SYSTEM Skills
  (* Version 1.0, 2019-10-15, dorofeev *)
  APPLICATION SkillsApp
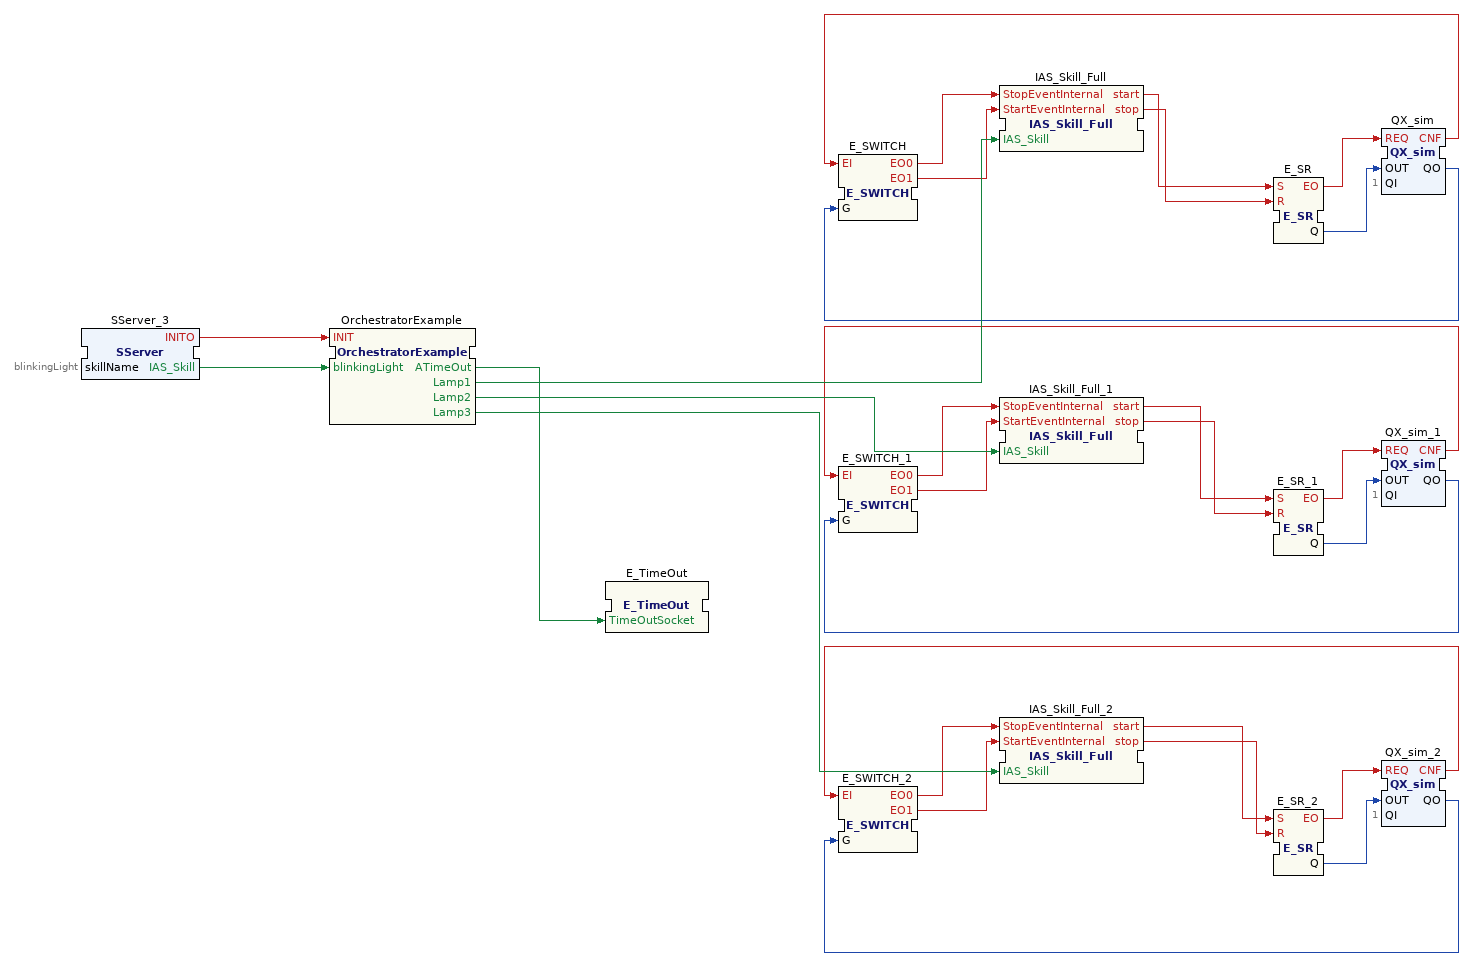
    FBS
      IAS_Skill_Full : IAS_Skill_Full;
      E_SR : E_SR;
      E_SWITCH : E_SWITCH;
      IAS_Skill_Full_1 : IAS_Skill_Full;
      E_SR_1 : E_SR;
      E_SWITCH_1 : E_SWITCH;
      IAS_Skill_Full_2 : IAS_Skill_Full;
      E_SR_2 : E_SR;
      E_SWITCH_2 : E_SWITCH;
      E_TimeOut : E_TimeOut;
      OrchestratorExample : OrchestratorExample;
    END_FBS
    SUBAPPS
      QX_sim : QX_sim(QI := 1);
      QX_sim_1 : QX_sim(QI := 1);
      QX_sim_2 : QX_sim(QI := 1);
      SServer_3 : SServer(skillName := blinkingLight);
    END_SUBAPPS
    EVENT_CONNECTIONS
      IAS_Skill_Full.start TO E_SR.S;
      IAS_Skill_Full.stop TO E_SR.R;
      E_SR.EO TO QX_sim.REQ;
      QX_sim.CNF TO E_SWITCH.EI;
      E_SWITCH.EO0 TO IAS_Skill_Full.StopEventInternal;
      E_SWITCH.EO1 TO IAS_Skill_Full.StartEventInternal;
      IAS_Skill_Full_1.start TO E_SR_1.S;
      E_SWITCH_1.EO0 TO IAS_Skill_Full_1.StopEventInternal;
      IAS_Skill_Full_1.stop TO E_SR_1.R;
      E_SWITCH_1.EO1 TO IAS_Skill_Full_1.StartEventInternal;
      QX_sim_1.CNF TO E_SWITCH_1.EI;
      E_SR_1.EO TO QX_sim_1.REQ;
      IAS_Skill_Full_2.start TO E_SR_2.S;
      E_SWITCH_2.EO0 TO IAS_Skill_Full_2.StopEventInternal;
      IAS_Skill_Full_2.stop TO E_SR_2.R;
      E_SWITCH_2.EO1 TO IAS_Skill_Full_2.StartEventInternal;
      QX_sim_2.CNF TO E_SWITCH_2.EI;
      E_SR_2.EO TO QX_sim_2.REQ;
      SServer_3.INITO TO OrchestratorExample.INIT;
    END_CONNECTIONS
    DATA_CONNECTIONS
      E_SR.Q TO QX_sim.OUT;
      QX_sim.QO TO E_SWITCH.G;
      E_SR_1.Q TO QX_sim_1.OUT;
      QX_sim_1.QO TO E_SWITCH_1.G;
      E_SR_2.Q TO QX_sim_2.OUT;
      QX_sim_2.QO TO E_SWITCH_2.G;
    END_CONNECTIONS
    ADAPTER_CONNECTIONS
      OrchestratorExample.ATimeOut TO E_TimeOut.TimeOutSocket;
      SServer_3.IAS_Skill TO OrchestratorExample.blinkingLight;
      OrchestratorExample.Lamp1 TO IAS_Skill_Full.IAS_Skill;
      OrchestratorExample.Lamp2 TO IAS_Skill_Full_1.IAS_Skill;
      OrchestratorExample.Lamp3 TO IAS_Skill_Full_2.IAS_Skill;
    END_CONNECTIONS
  END_APPLICATION
  APPLICATION test
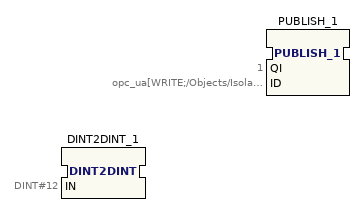
    FBS
      PUBLISH_1 : PUBLISH_1(QI := 1, ID := opc_ua[WRITE;/Objects/IsolatedTests/WRITEVariable]);
      DINT2DINT_1 : DINT2DINT(IN := DINT#12);
    END_FBS
  END_APPLICATION
  DEVICE skillConsumer : FORTE_PC(MGR_ID := "localhost:61499")
    {SET_ATTRIBUTE(Profile, HOLOBLOC)} (* device profile *)
    RESOURCE EMB_RES : EMB_RES
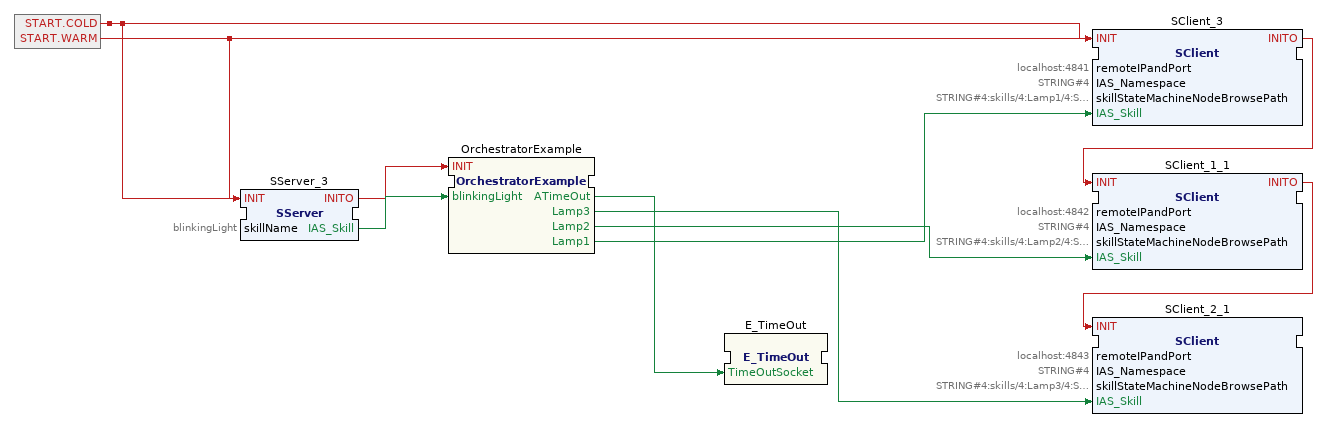
      FBS
        E_TimeOut : E_TimeOut;
        OrchestratorExample : OrchestratorExample;
      END_FBS
      SUBAPPS
        SServer_3 : SServer(skillName := blinkingLight);
        SClient_2_1 : SClient(remoteIPandPort := localhost:4843, IAS_Namespace := STRING#4, skillStateMachineNodeBrowsePath := STRING#4:skills/4:Lamp3/4:StateMachine/);
        SClient_3 : SClient(remoteIPandPort := localhost:4841, IAS_Namespace := STRING#4, skillStateMachineNodeBrowsePath := STRING#4:skills/4:Lamp1/4:StateMachine/);
        SClient_1_1 : SClient(remoteIPandPort := localhost:4842, IAS_Namespace := STRING#4, skillStateMachineNodeBrowsePath := STRING#4:skills/4:Lamp2/4:StateMachine/);
      END_SUBAPPS
      EVENT_CONNECTIONS
        SServer_3.INITO TO OrchestratorExample.INIT;
        START.COLD TO SServer_3.INIT;
        START.WARM TO SServer_3.INIT;
        SClient_1_1.INITO TO SClient_2_1.INIT;
        SClient_3.INITO TO SClient_1_1.INIT;
        START.COLD TO SClient_3.INIT;
        START.WARM TO SClient_3.INIT;
      END_CONNECTIONS
      ADAPTER_CONNECTIONS
        OrchestratorExample.ATimeOut TO E_TimeOut.TimeOutSocket;
        SServer_3.IAS_Skill TO OrchestratorExample.blinkingLight;
        OrchestratorExample.Lamp3 TO SClient_2_1.IAS_Skill;
        OrchestratorExample.Lamp2 TO SClient_1_1.IAS_Skill;
        OrchestratorExample.Lamp1 TO SClient_3.IAS_Skill;
      END_CONNECTIONS
    END_RESOURCE
  END_DEVICE
  DEVICE skillProvider1 : FORTE_PC(MGR_ID := "localhost:61500")
    {SET_ATTRIBUTE(Profile, HOLOBLOC)} (* device profile *)
    RESOURCE EMB_RES : EMB_RES
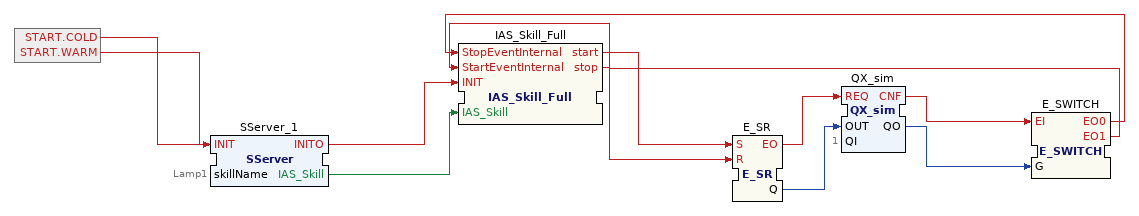
      FBS
        IAS_Skill_Full : IAS_Skill_Full;
        E_SWITCH : E_SWITCH;
        E_SR : E_SR;
      END_FBS
      SUBAPPS
        QX_sim : QX_sim(QI := 1);
        SServer_1 : SServer(skillName := Lamp1);
      END_SUBAPPS
      EVENT_CONNECTIONS
        QX_sim.CNF TO E_SWITCH.EI;
        E_SWITCH.EO0 TO IAS_Skill_Full.StopEventInternal;
        E_SWITCH.EO1 TO IAS_Skill_Full.StartEventInternal;
        IAS_Skill_Full.start TO E_SR.S;
        IAS_Skill_Full.stop TO E_SR.R;
        E_SR.EO TO QX_sim.REQ;
        START.COLD TO SServer_1.INIT;
        START.WARM TO SServer_1.INIT;
        SServer_1.INITO TO IAS_Skill_Full.INIT;
      END_CONNECTIONS
      DATA_CONNECTIONS
        QX_sim.QO TO E_SWITCH.G;
        E_SR.Q TO QX_sim.OUT;
      END_CONNECTIONS
      ADAPTER_CONNECTIONS
        SServer_1.IAS_Skill TO IAS_Skill_Full.IAS_Skill;
      END_CONNECTIONS
    END_RESOURCE
  END_DEVICE
  DEVICE skillProvider2 : FORTE_PC(MGR_ID := "localhost:61501")
    {SET_ATTRIBUTE(Profile, HOLOBLOC)} (* device profile *)
    RESOURCE EMB_RES : EMB_RES
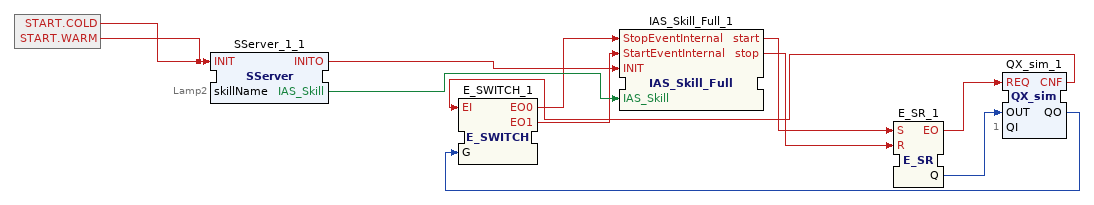
      FBS
        IAS_Skill_Full_1 : IAS_Skill_Full;
        E_SR_1 : E_SR;
        E_SWITCH_1 : E_SWITCH;
      END_FBS
      SUBAPPS
        QX_sim_1 : QX_sim(QI := 1);
        SServer_1_1 : SServer(skillName := Lamp2);
      END_SUBAPPS
      EVENT_CONNECTIONS
        IAS_Skill_Full_1.start TO E_SR_1.S;
        IAS_Skill_Full_1.stop TO E_SR_1.R;
        E_SR_1.EO TO QX_sim_1.REQ;
        QX_sim_1.CNF TO E_SWITCH_1.EI;
        E_SWITCH_1.EO0 TO IAS_Skill_Full_1.StopEventInternal;
        E_SWITCH_1.EO1 TO IAS_Skill_Full_1.StartEventInternal;
        START.COLD TO SServer_1_1.INIT;
        START.WARM TO SServer_1_1.INIT;
        SServer_1_1.INITO TO IAS_Skill_Full_1.INIT;
      END_CONNECTIONS
      DATA_CONNECTIONS
        E_SR_1.Q TO QX_sim_1.OUT;
        QX_sim_1.QO TO E_SWITCH_1.G;
      END_CONNECTIONS
      ADAPTER_CONNECTIONS
        SServer_1_1.IAS_Skill TO IAS_Skill_Full_1.IAS_Skill;
      END_CONNECTIONS
    END_RESOURCE
  END_DEVICE
  DEVICE skillProvider3 : FORTE_PC(MGR_ID := "localhost:61502")
    {SET_ATTRIBUTE(Profile, HOLOBLOC)} (* device profile *)
    RESOURCE EMB_RES : EMB_RES
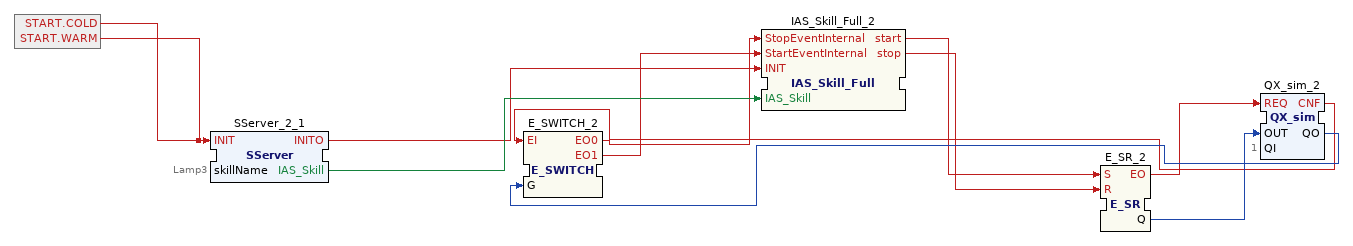
      FBS
        E_SWITCH_2 : E_SWITCH;
        E_SR_2 : E_SR;
        IAS_Skill_Full_2 : IAS_Skill_Full;
      END_FBS
      SUBAPPS
        QX_sim_2 : QX_sim(QI := 1);
        SServer_2_1 : SServer(skillName := Lamp3);
      END_SUBAPPS
      EVENT_CONNECTIONS
        E_SR_2.EO TO QX_sim_2.REQ;
        QX_sim_2.CNF TO E_SWITCH_2.EI;
        E_SWITCH_2.EO0 TO IAS_Skill_Full_2.StopEventInternal;
        E_SWITCH_2.EO1 TO IAS_Skill_Full_2.StartEventInternal;
        IAS_Skill_Full_2.start TO E_SR_2.S;
        IAS_Skill_Full_2.stop TO E_SR_2.R;
        START.COLD TO SServer_2_1.INIT;
        START.WARM TO SServer_2_1.INIT;
        SServer_2_1.INITO TO IAS_Skill_Full_2.INIT;
      END_CONNECTIONS
      DATA_CONNECTIONS
        E_SR_2.Q TO QX_sim_2.OUT;
        QX_sim_2.QO TO E_SWITCH_2.G;
      END_CONNECTIONS
      ADAPTER_CONNECTIONS
        SServer_2_1.IAS_Skill TO IAS_Skill_Full_2.IAS_Skill;
      END_CONNECTIONS
    END_RESOURCE
  END_DEVICE
  MAPPINGS
    SkillsApp.IAS_Skill_Full ON skillProvider1.EMB_RES.IAS_Skill_Full;
    SkillsApp.QX_sim ON skillProvider1.EMB_RES.QX_sim;
    SkillsApp.E_SWITCH ON skillProvider1.EMB_RES.E_SWITCH;
    SkillsApp.E_SR ON skillProvider1.EMB_RES.E_SR;
    SkillsApp.IAS_Skill_Full_1 ON skillProvider2.EMB_RES.IAS_Skill_Full_1;
    SkillsApp.E_SR_1 ON skillProvider2.EMB_RES.E_SR_1;
    SkillsApp.QX_sim_1 ON skillProvider2.EMB_RES.QX_sim_1;
    SkillsApp.E_SWITCH_1 ON skillProvider2.EMB_RES.E_SWITCH_1;
    SkillsApp.E_SWITCH_2 ON skillProvider3.EMB_RES.E_SWITCH_2;
    SkillsApp.E_SR_2 ON skillProvider3.EMB_RES.E_SR_2;
    SkillsApp.QX_sim_2 ON skillProvider3.EMB_RES.QX_sim_2;
    SkillsApp.IAS_Skill_Full_2 ON skillProvider3.EMB_RES.IAS_Skill_Full_2;
    SkillsApp.E_TimeOut ON skillConsumer.EMB_RES.E_TimeOut;
    SkillsApp.OrchestratorExample ON skillConsumer.EMB_RES.OrchestratorExample;
    SkillsApp.SServer_3 ON skillConsumer.EMB_RES.SServer_3;
  END_MAPPINGS
  SEGMENTS
    Ethernet : Ethernet;
  END_SEGMENTS
  LINKS
    skillConsumer => Ethernet;
    skillProvider1 => Ethernet;
    skillProvider2 => Ethernet;
    skillProvider3 => Ethernet;
  END_LINKS
END_SYSTEM
